// Function block for AC motors controlled with the LENZE d-31855 frequency inverter
FUNCTION_BLOCK FB_Component_ACmotor IMPLEMENTS I_Component
VAR_INPUT
	bDeviceActive	: BOOL; // relay contact freq inv
	// Interface vars
	sName			: STRING[20];
	bEnable     	: BOOL;
	//eMode       	: E_ComponentMode;
END_VAR

VAR_OUTPUT
	eJogFreq		: E_LenzeJogFreq := E_LenzeJogFreq.F0FF;
	// interface vars	
	eState			: E_State;
	iErrorCode		: INT;
	sStatusText 	: STRING[50];
END_VAR

VAR_IN_OUT
	bE1jog1			: BOOL;					// jog func b1
	bE2jog2			: BOOL;					// jog func b2
	bE3DCbrake		: BOOL;					// DC injection brake
	eE4Direction	: BOOL;	// motor direction
END_VAR

IF bDeviceActive AND bEnable AND (eState = E_State.READY OR eState = E_State.BUSY) THEN
	// set jog frequency
	CASE eJogFreq OF
		E_LenzeJogFreq.F0FF: 	bE1jog1 	:= FALSE;
								bE2jog2 	:= FALSE;
								//bE3DCbrake 	:= TRUE;
								eState		:= E_State.READY;
		E_LenzeJogFreq.F1: 		bE1jog1 	:= TRUE;
								bE2jog2 	:= FALSE;
								//bE3DCbrake 	:= FALSE;
								eState		:= E_State.BUSY;
		E_LenzeJogFreq.F2: 		bE1jog1 	:= TRUE;
								bE2jog2 	:= TRUE;
								//bE3DCbrake 	:= FALSE;
								eState		:= E_State.BUSY;
		E_LenzeJogFreq.F3: 		bE1jog1 	:= FALSE;
								bE2jog2 	:= TRUE;
								//bE3DCbrake 	:= FALSE;
								eState		:= E_State.BUSY;
	END_CASE

ELSE
	bE1jog1 := FALSE;
	bE2jog2 := FALSE;
	eState	:= E_State.READY;
END_IF

METHOD M_Halt : BOOL
bE1jog1 := FALSE;
bE2jog2 := FALSE;
eState := E_State.HALTED;
END_METHOD

METHOD M_SetDir : BOOL
VAR_INPUT
	Direction: E_RotationDirection;
END_VAR
eE4Direction := TO_BOOL(Direction);
END_METHOD

METHOD M_SetFreq : BOOL
VAR_INPUT
	Frequency: E_LenzeJogFreq;
END_VAR
eJogFreq := Frequency;
END_METHOD

METHOD M_Start : BOOL
IF eState <> E_State.BUSY THEN
	eState := E_State.READY;
END_IF;
END_METHOD

METHOD M_Stop : BOOL
IF eState <> E_State.BUSY THEN
	bE1jog1 := FALSE;
	bE2jog2 := FALSE;	
	eState := E_State.DONE;
END_IF
END_METHOD

END_FUNCTION_BLOCK

(* stored: Version 1.1.0.1, ProductVersion 3.1.4024.15
   POU FB_Component_ACmotor: Id {4bee0a47-7e8d-4a20-bf36-74643afc4427}, SpecialFunc None
   Method M_Halt: Id {86f47aa8-e6c4-4e8a-ae11-d7c42ced5250}
   Method M_SetDir: Id {d6a197ac-aaf3-4f2e-919c-b2334f169d78}
   Method M_SetFreq: Id {387ee47f-c4da-4cf1-a6b6-e28ea3f37257}
   Method M_Start: Id {8c2f0a58-166c-44b6-b1c3-800306693fc7}
   Method M_Stop: Id {84392872-6e4d-4fd5-a526-059b31207e24} *)
